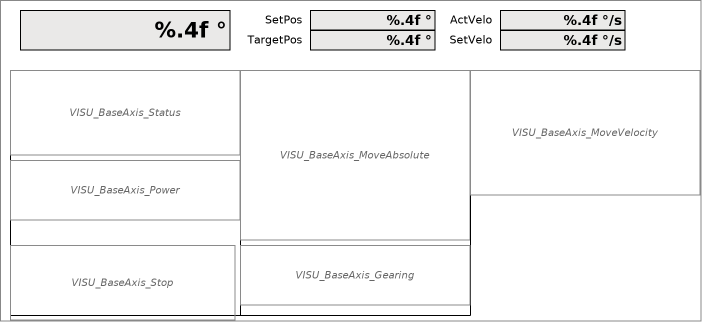
VISUALIZATION VISU_AngularAxis  // 702x322
VAR_IN_OUT
	axis : AngularAxis;
	widget : AngularAxisWidget;
END_VAR
    Rectangle (20,10 210x40), "%.4f °", text variable: axis.actPos.degrees.value
    Line (240,80) (240,315)
    Line (10,80) (10,315)
    Line (10,315) (470,315)
    Frame (10,70 230x85)
        shows VISU_BaseAxis_Status(axis := axis, axisWidget := widget.base)
    Frame (10,160 230x60)
        shows VISU_BaseAxis_Power(axis := axis, axisWidget := widget.base)
    Frame (240,70 230x170)
        shows VISU_BaseAxis_MoveAbsolute(axis := axis, axisWidget := widget.base, positionSymbol := widget.positionSymbol, velocitySymbol := widget.velocitySymbol)
    Frame (10,245 225x75)
        shows VISU_BaseAxis_Stop(axis := axis, axisWidget := widget.base)
    Line (470,80) (470,315)
    Frame (240,245 230x60)
        shows VISU_BaseAxis_Gearing(axis := axis, axisWidget := widget.base)
    Frame (470,70 230x125)
        shows VISU_BaseAxis_MoveVelocity(axis := axis, axisWidget := widget.base, positionSymbol := widget.positionSymbol, velocitySymbol := widget.velocitySymbol)
    Rectangle (310,10 125x20), "%.4f °", text variable: axis.axis_ref.NcToPlc.SetPos
    Label (255,10 50x20), "SetPos"
    Rectangle (310,30 125x20), "%.4f °", text variable: axis.axis_ref.NcToPlc.TargetPos
    Label (240,30 65x20), "TargetPos"
    Rectangle (500,10 125x20), "%.4f °/s", text variable: axis.axis_ref.NcToPlc.ActVelo
    Label (445,10 50x20), "ActVelo"
    Label (445,30 50x20), "SetVelo"
    Rectangle (500,30 125x20), "%.4f °/s", text variable: axis.axis_ref.NcToPlc.SetVelo
END_VISUALIZATION

(* stored: Version 1.1.0.1, ProductVersion 3.1.4019.2
   Visu VISU_AngularAxis: Id {7406a597-2320-4b6e-8ff3-5ff0f461717f} *)
